// TIA Portal V20 export
// export: Created 2025-12-01T14:57:24.1509641Z, ExportSetting None, DisplayName Totally Integrated Automation Portal, DisplayVersion V20 Update 3, DisplayName TIA Portal Openness, DisplayVersion V20 Update 3, DisplayName TIA Portal Version Control Interface, DisplayVersion V20 Update 3, DisplayName STEP 7 Professional, DisplayVersion V20 Update 3, DisplayName STEP 7 Safety, DisplayVersion V20 Update 2, DisplayName WinCC Basic/Comfort/Advanced, DisplayVersion V20 Update 3, DisplayName WinCC Professional, DisplayVersion V20 Update 3, DisplayName WinCC Unified, DisplayVersion V20 Update 3
FUNCTION "FC960_ScadaMesa" : Void   // FC960, STL
TITLE = Funcion de Tratamiento de la Mesa para el SCADA
{ S7_Optimized_Access := 'FALSE' }
AUTHOR : SCADA
NAME : 20160901
VERSION : 1.0
// stored: AutoNumber false
   VAR_INPUT
      NumMesa : UInt;
   END_VAR
   VAR_TEMP
      Mesa : UInt;
      EnMarcha : Bool;
      EnError : Bool;
   END_VAR
BEGIN

NETWORK
TITLE = Inicializacion
//////////////////////////////////////////////////////////////////////////////
//////////////////////////////////////////////////////////////////////////////
/// Tareas Iniciales de Inicializacion

      L     #NumMesa;  // Numero de Mesa a tratar
      T     #Mesa;



NETWORK
TITLE = Contadores de Flujos
//////////////////////////////////////////////////////////////////////////////
//////////////////////////////////////////////////////////////////////////////
/// Calculo de Bultos Totales

/// -- Bultos Entrada Totales Carga E0 + E1 + E2 + E3 + E4
      SET;
      A     "DB900_Estado_Mesas".EstadoVI[#Mesa].Etapas_Carga_E0;
      O     "DB900_Estado_Mesas".EstadoVI[#Mesa].Etapas_Carga_E1;
      O     "DB900_Estado_Mesas".EstadoVI[#Mesa].Etapas_Carga_E2;
      O     "DB900_Estado_Mesas".EstadoVI[#Mesa].Etapas_Carga_E3;
      O     "DB900_Estado_Mesas".EstadoVI[#Mesa].Etapas_Carga_E4;
      FP    "DB011_ScadaMesas".Mesa[#Mesa].MemoBultos_Totales;
      JCN   NBTO;  // Una entrada mas ?

      L     "DB011_ScadaMesas".Mesa[#Mesa].Bultos_Totales;  // +1
      L     1;
      +I;
      T     "DB011_ScadaMesas".Mesa[#Mesa].Bultos_Totales;

NBTO: NOP   0;



NETWORK
TITLE = ---
//////////////////////////////////////////////////////////////////////////////
//////////////////////////////////////////////////////////////////////////////
/// Calculo de Bultos de Entrada

/// -- Bultos de Entrada por E1
      SET;
      A     "DB900_Estado_Mesas".EstadoVI[#Mesa].Etapas_Carga_E1;
      FP    "DB011_ScadaMesas".Mesa[#Mesa].MemoBultos_E1;
      JCN   NBE1;  // Una entrada mas ?

      L     "DB011_ScadaMesas".Mesa[#Mesa].Bultos_E1;  // +1
      L     1;
      +I;
      T     "DB011_ScadaMesas".Mesa[#Mesa].Bultos_E1;

NBE1: NOP   0;


/// -- Bultos de Entrada por E2
      SET;
      A     "DB900_Estado_Mesas".EstadoVI[#Mesa].Etapas_Carga_E2;
      FP    "DB011_ScadaMesas".Mesa[#Mesa].MemoBultos_E2;
      JCN   NBE2;  // Una entrada mas ?

      L     "DB011_ScadaMesas".Mesa[#Mesa].Bultos_E2;  // +1
      L     1;
      +I;
      T     "DB011_ScadaMesas".Mesa[#Mesa].Bultos_E2;

NBE2: NOP   0;


/// -- Bultos de Entrada por E3
      SET;
      A     "DB900_Estado_Mesas".EstadoVI[#Mesa].Etapas_Carga_E3;
      FP    "DB011_ScadaMesas".Mesa[#Mesa].MemoBultos_E3;
      JCN   NBE3;  // Una entrada mas ?

      L     "DB011_ScadaMesas".Mesa[#Mesa].Bultos_E3;  // +1
      L     1;
      +I;
      T     "DB011_ScadaMesas".Mesa[#Mesa].Bultos_E3;

NBE3: NOP   0;


/// -- Bultos de Entrada por E4
      SET;
      A     "DB900_Estado_Mesas".EstadoVI[#Mesa].Etapas_Carga_E4;
      FP    "DB011_ScadaMesas".Mesa[#Mesa].MemoBultos_E4;
      JCN   NBE4;  // Una entrada mas ?

      L     "DB011_ScadaMesas".Mesa[#Mesa].Bultos_E4;  // +1
      L     1;
      +I;
      T     "DB011_ScadaMesas".Mesa[#Mesa].Bultos_E4;

NBE4: NOP   0;



NETWORK
TITLE = ---
//////////////////////////////////////////////////////////////////////////////
//////////////////////////////////////////////////////////////////////////////
/// Calculo de Bultos de Salida

/// -- Bultos de Salida por S1
      SET;
      A     "DB900_Estado_Mesas".EstadoVI[#Mesa].Etapas_Descarga_S1;
      FP    "DB011_ScadaMesas".Mesa[#Mesa].MemoBultos_S1;
      JCN   NBS1;  // Una entrada mas ?

      L     "DB011_ScadaMesas".Mesa[#Mesa].Bultos_S1;  // +1
      L     1;
      +I;
      T     "DB011_ScadaMesas".Mesa[#Mesa].Bultos_S1;

NBS1: NOP   0;


// ---- Bultos de Salida por S2
      SET;
      A     "DB900_Estado_Mesas".EstadoVI[#Mesa].Etapas_Descarga_S2;
      FP    "DB011_ScadaMesas".Mesa[#Mesa].MemoBultos_S2;
      JCN   NBS2;  // Una entrada mas ?

      L     "DB011_ScadaMesas".Mesa[#Mesa].Bultos_S2;  // +1
      L     1;
      +I;
      T     "DB011_ScadaMesas".Mesa[#Mesa].Bultos_S2;

NBS2: NOP   0;


// ---- Bultos de Salida por S3
      SET;
      A     "DB900_Estado_Mesas".EstadoVI[#Mesa].Etapas_Descarga_S3;
      FP    "DB011_ScadaMesas".Mesa[#Mesa].MemoBultos_S3;
      JCN   NBS3;  // Una entrada mas ?

      L     "DB011_ScadaMesas".Mesa[#Mesa].Bultos_S3;  // +1
      L     1;
      +I;
      T     "DB011_ScadaMesas".Mesa[#Mesa].Bultos_S3;

NBS3: NOP   0;


// ---- Bultos de Salida por S4
      SET;
      A     "DB900_Estado_Mesas".EstadoVI[#Mesa].Etapas_Descarga_S4;
      FP    "DB011_ScadaMesas".Mesa[#Mesa].MemoBultos_S4;
      JCN   NBS4;  // Una entrada mas ?

      L     "DB011_ScadaMesas".Mesa[#Mesa].Bultos_S4;  // +1
      L     1;
      +I;
      T     "DB011_ScadaMesas".Mesa[#Mesa].Bultos_S4;

NBS4: NOP   0;




NETWORK
TITLE = Tiempo de Fallo
//////////////////////////////////////////////////////////////////////////////
//////////////////////////////////////////////////////////////////////////////
/// Calculo de Tiempo En Fallo
      SET;
      A     "DB900_Estado_Mesas".EstadoVI[#Mesa].Error_Mx;
      =     #EnError;

      SET;
      AN    #EnError;  // Contar Tiempo ?
      JC    N_ER;

      CALL  "FC914_SumaTiempo_DT"
      ( TiempoActual := "DB011_ScadaMesas".Mesa[#Mesa].TMP_Error
      );

N_ER: NOP   0;



NETWORK
TITLE = Informacion de los Motores
//////////////////////////////////////////////////////////////////////////////
//////////////////////////////////////////////////////////////////////////////
/// Calculo de Arranques

/// -- Numero de Arranques del M1 // Rodillos Avance y Retroceso
      SET;
      A     "DB900_Estado_Mesas".EstadoVI[#Mesa].Sa_Rod_Avance;
      O     "DB900_Estado_Mesas".EstadoVI[#Mesa].Sa_Rod_Retroc;
      FP    "DB011_ScadaMesas".Mesa[#Mesa].MemoArranques_M1;
      JCN   NAM1;  // Un arranque Mas mas ?

      L     "DB011_ScadaMesas".Mesa[#Mesa].Arranques_M1;  // +1
      L     1;
      +I;
      T     "DB011_ScadaMesas".Mesa[#Mesa].Arranques_M1;

NAM1: NOP   0;


/// -- Numero de Arranques del M2 // Cadenas Avance y Retroceso
      SET;
      A     "DB900_Estado_Mesas".EstadoVI[#Mesa].Sa_Cad_Avance;
      O     "DB900_Estado_Mesas".EstadoVI[#Mesa].Sa_Cad_Retroc;
      FP    "DB011_ScadaMesas".Mesa[#Mesa].MemoArranques_M2;
      JCN   NAM2;  // Un arranque Mas mas ?

      L     "DB011_ScadaMesas".Mesa[#Mesa].Arranques_M2;  // +1
      L     1;
      +I;
      T     "DB011_ScadaMesas".Mesa[#Mesa].Arranques_M2;

NAM2: NOP   0;


/// -- Numero de Arranques del M3 // Giro Derechas y Izaquierdas
      SET;
      A     "DB900_Estado_Mesas".EstadoVI[#Mesa].Sa_Giro_0;
      O     "DB900_Estado_Mesas".EstadoVI[#Mesa].Sa_Giro_90;
      FP    "DB011_ScadaMesas".Mesa[#Mesa].MemoArranques_M3;
      JCN   NAM3;  // Un arranque Mas mas ?

      L     "DB011_ScadaMesas".Mesa[#Mesa].Arranques_M3;  // +1
      L     1;
      +I;
      T     "DB011_ScadaMesas".Mesa[#Mesa].Arranques_M3;

NAM3: NOP   0;


/// -- Numero de Arranques del M4 // Subir y Bajar Transfer
      SET;
      A     "DB900_Estado_Mesas".EstadoVI[#Mesa].Sa_Trans_Sub;
      O     "DB900_Estado_Mesas".EstadoVI[#Mesa].Sa_Trans_Baj;
      FP    "DB011_ScadaMesas".Mesa[#Mesa].MemoArranques_M4;
      JCN   NAM4;  // Un arranque Mas mas ?

      L     "DB011_ScadaMesas".Mesa[#Mesa].Arranques_M4;  // +1
      L     1;
      +I;
      T     "DB011_ScadaMesas".Mesa[#Mesa].Arranques_M4;

NAM4: NOP   0;


/// -- Numero de Arranques del M5 // Subir y Bajar Tope
      SET;
      A     "DB900_Estado_Mesas".EstadoVI[#Mesa].Sa_Tope1_Sub;
      O     "DB900_Estado_Mesas".EstadoVI[#Mesa].Sa_Tope1_Baj;
      FP    "DB011_ScadaMesas".Mesa[#Mesa].MemoArranques_M5;
      JCN   NAM5;  // Un arranque Mas mas ?

      L     "DB011_ScadaMesas".Mesa[#Mesa].Arranques_M5;  // +1
      L     1;
      +I;
      T     "DB011_ScadaMesas".Mesa[#Mesa].Arranques_M5;

NAM5: NOP   0;



NETWORK
TITLE = ---
// --------------------------------------------------------------------------------------------------
// --------------------------------------------------------------------------------------------------
// --- Calculo de Tiempo

/// -- Tiempo en Marcha M1 // Rodillos Avance y Retroceso
      SET;
      A     "DB900_Estado_Mesas".EstadoVI[#Mesa].Sa_Rod_Avance;
      O     "DB900_Estado_Mesas".EstadoVI[#Mesa].Sa_Rod_Retroc;
      =     #EnMarcha;

      SET;
      AN    #EnMarcha;  // Contar Tiempo ?
      JC    N_M1;

      CALL  "FC914_SumaTiempo_DT"
      ( TiempoActual := "DB011_ScadaMesas".Mesa[#Mesa].TMP_Marcha_M1
      );

N_M1: NOP   0;


/// -- Tiempo en Marcha M2 // Cadenas Avance y Retroceso
      SET;
      A     "DB900_Estado_Mesas".EstadoVI[#Mesa].Sa_Cad_Avance;
      O     "DB900_Estado_Mesas".EstadoVI[#Mesa].Sa_Cad_Retroc;
      =     #EnMarcha;

      SET;
      AN    #EnMarcha;  // Contar Tiempo ?
      JC    N_M2;

      CALL  "FC914_SumaTiempo_DT"
      ( TiempoActual := "DB011_ScadaMesas".Mesa[#Mesa].TMP_Marcha_M2
      );

N_M2: NOP   0;


/// -- Tiempo en Marcha M3 //Giro Derechas y Izaquierdas
      SET;
      A     "DB900_Estado_Mesas".EstadoVI[#Mesa].Sa_Giro_0;
      O     "DB900_Estado_Mesas".EstadoVI[#Mesa].Sa_Giro_90;
      =     #EnMarcha;

      SET;
      AN    #EnMarcha;  // Contar Tiempo ?
      JC    N_M3;

      CALL  "FC914_SumaTiempo_DT"
      ( TiempoActual := "DB011_ScadaMesas".Mesa[#Mesa].TMP_Marcha_M3
      );

N_M3: NOP   0;


// ---- Tiempo en Marcha M4 // Subir y Bajar Transfer
      SET;
      A     "DB900_Estado_Mesas".EstadoVI[#Mesa].Sa_Trans_Sub;
      O     "DB900_Estado_Mesas".EstadoVI[#Mesa].Sa_Trans_Baj;
      =     #EnMarcha;

      SET;
      AN    #EnMarcha;  // Contar Tiempo ?
      JC    N_M4;

      CALL  "FC914_SumaTiempo_DT"
      ( TiempoActual := "DB011_ScadaMesas".Mesa[#Mesa].TMP_Marcha_M4
      );

N_M4: NOP   0;


// ---- Tiempo en Marcha M5 // Subir y Bajar Tope
      SET;
      A     "DB900_Estado_Mesas".EstadoVI[#Mesa].Sa_Tope1_Sub;
      O     "DB900_Estado_Mesas".EstadoVI[#Mesa].Sa_Tope1_Baj;
      =     #EnMarcha;

      SET;
      AN    #EnMarcha;  // Contar Tiempo ?
      JC    N_M5;

      CALL  "FC914_SumaTiempo_DT"
      ( TiempoActual := "DB011_ScadaMesas".Mesa[#Mesa].TMP_Marcha_M5
      );

N_M5: NOP   0;



NETWORK
TITLE = Final de la Funcion
//////////////////////////////////////////////////////////////////////////////
//////////////////////////////////////////////////////////////////////////////
/// Tareas de Finalizacion de la Funcion


END_FUNCTION
